Universal Robots URScript: quanser_2_150.script

def initialization():
	global program_counter = 1
end
def main():
	first_trajectory_pose = pose_inv(p[0.6, 0.0, 0.617008797653959, -1.20919957615615, 1.20919957615615, -1.20919957615615])
	starting_pose_tcp = get_actual_tcp_pose()
	counter = 0
while(counter < program_counter):
	movel(pose_trans(starting_pose_tcp, pose_trans(first_trajectory_pose,p[0.55, 0.0, 0.617008797653959, -1.20919957615615, 1.20919957615615, -1.20919957615615])), r=0.0)
	movel(pose_trans(starting_pose_tcp, pose_trans(first_trajectory_pose,p[0.55, 0.00146627565982405, 0.401466275659824, -1.20919957615615, 1.20919957615615, -1.20919957615615])), r=0.0)
	movel(pose_trans(starting_pose_tcp, pose_trans(first_trajectory_pose,p[0.6, 0.00146627565982405, 0.401466275659824, -1.20919957615615, 1.20919957615615, -1.20919957615615])), r=0.0)
	movel(pose_trans(starting_pose_tcp, pose_trans(first_trajectory_pose,p[0.6, 0.00879765395894428, 0.401466275659824, -1.20919957615615, 1.20919957615615, -1.20919957615615])), r=0.0)
	movel(pose_trans(starting_pose_tcp, pose_trans(first_trajectory_pose,p[0.6, 0.0161290322580645, 0.401466275659824, -1.20919957615615, 1.20919957615615, -1.20919957615615])), r=0.0)
	movel(pose_trans(starting_pose_tcp, pose_trans(first_trajectory_pose,p[0.6, 0.0234604105571848, 0.401466275659824, -1.20919957615615, 1.20919957615615, -1.20919957615615])), r=0.0)
	movel(pose_trans(starting_pose_tcp, pose_trans(first_trajectory_pose,p[0.6, 0.030791788856305, 0.401466275659824, -1.20919957615615, 1.20919957615615, -1.20919957615615])), r=0.0)
	movel(pose_trans(starting_pose_tcp, pose_trans(first_trajectory_pose,p[0.6, 0.0381231671554252, 0.401466275659824, -1.20919957615615, 1.20919957615615, -1.20919957615615])), r=0.0)
	movel(pose_trans(starting_pose_tcp, pose_trans(first_trajectory_pose,p[0.6, 0.0454545454545455, 0.401466275659824, -1.20919957615615, 1.20919957615615, -1.20919957615615])), r=0.0)
	movel(pose_trans(starting_pose_tcp, pose_trans(first_trajectory_pose,p[0.6, 0.0527859237536657, 0.401466275659824, -1.20919957615615, 1.20919957615615, -1.20919957615615])), r=0.0)
	movel(pose_trans(starting_pose_tcp, pose_trans(first_trajectory_pose,p[0.6, 0.0601173020527859, 0.401466275659824, -1.20919957615615, 1.20919957615615, -1.20919957615615])), r=0.0)
	movel(pose_trans(starting_pose_tcp, pose_trans(first_trajectory_pose,p[0.6, 0.0674486803519062, 0.401466275659824, -1.20919957615615, 1.20919957615615, -1.20919957615615])), r=0.0)
	movel(pose_trans(starting_pose_tcp, pose_trans(first_trajectory_pose,p[0.6, 0.0747800586510264, 0.401466275659824, -1.20919957615615, 1.20919957615615, -1.20919957615615])), r=0.0)
	movel(pose_trans(starting_pose_tcp, pose_trans(first_trajectory_pose,p[0.6, 0.0821114369501466, 0.401466275659824, -1.20919957615615, 1.20919957615615, -1.20919957615615])), r=0.0)
	movel(pose_trans(starting_pose_tcp, pose_trans(first_trajectory_pose,p[0.6, 0.0894428152492669, 0.401466275659824, -1.20919957615615, 1.20919957615615, -1.20919957615615])), r=0.0)
	movel(pose_trans(starting_pose_tcp, pose_trans(first_trajectory_pose,p[0.6, 0.0967741935483871, 0.401466275659824, -1.20919957615615, 1.20919957615615, -1.20919957615615])), r=0.0)
	movel(pose_trans(starting_pose_tcp, pose_trans(first_trajectory_pose,p[0.6, 0.104105571847507, 0.401466275659824, -1.20919957615615, 1.20919957615615, -1.20919957615615])), r=0.0)
	movel(pose_trans(starting_pose_tcp, pose_trans(first_trajectory_pose,p[0.6, 0.111436950146628, 0.401466275659824, -1.20919957615615, 1.20919957615615, -1.20919957615615])), r=0.0)
	movel(pose_trans(starting_pose_tcp, pose_trans(first_trajectory_pose,p[0.6, 0.118768328445748, 0.401466275659824, -1.20919957615615, 1.20919957615615, -1.20919957615615])), r=0.0)
	movel(pose_trans(starting_pose_tcp, pose_trans(first_trajectory_pose,p[0.6, 0.126099706744868, 0.401466275659824, -1.20919957615615, 1.20919957615615, -1.20919957615615])), r=0.0)
	movel(pose_trans(starting_pose_tcp, pose_trans(first_trajectory_pose,p[0.6, 0.133431085043988, 0.401466275659824, -1.20919957615615, 1.20919957615615, -1.20919957615615])), r=0.0)
	movel(pose_trans(starting_pose_tcp, pose_trans(first_trajectory_pose,p[0.6, 0.140762463343109, 0.401466275659824, -1.20919957615615, 1.20919957615615, -1.20919957615615])), r=0.0)
	movel(pose_trans(starting_pose_tcp, pose_trans(first_trajectory_pose,p[0.6, 0.148093841642229, 0.401466275659824, -1.20919957615615, 1.20919957615615, -1.20919957615615])), r=0.0)
	movel(pose_trans(starting_pose_tcp, pose_trans(first_trajectory_pose,p[0.6, 0.155425219941349, 0.401466275659824, -1.20919957615615, 1.20919957615615, -1.20919957615615])), r=0.0)
	movel(pose_trans(starting_pose_tcp, pose_trans(first_trajectory_pose,p[0.6, 0.162756598240469, 0.401466275659824, -1.20919957615615, 1.20919957615615, -1.20919957615615])), r=0.0)
	movel(pose_trans(starting_pose_tcp, pose_trans(first_trajectory_pose,p[0.6, 0.170087976539589, 0.401466275659824, -1.20919957615615, 1.20919957615615, -1.20919957615615])), r=0.0)
	movel(pose_trans(starting_pose_tcp, pose_trans(first_trajectory_pose,p[0.6, 0.17741935483871, 0.401466275659824, -1.20919957615615, 1.20919957615615, -1.20919957615615])), r=0.0)
	movel(pose_trans(starting_pose_tcp, pose_trans(first_trajectory_pose,p[0.6, 0.18475073313783, 0.401466275659824, -1.20919957615615, 1.20919957615615, -1.20919957615615])), r=0.0)
	movel(pose_trans(starting_pose_tcp, pose_trans(first_trajectory_pose,p[0.6, 0.19208211143695, 0.401466275659824, -1.20919957615615, 1.20919957615615, -1.20919957615615])), r=0.0)
	movel(pose_trans(starting_pose_tcp, pose_trans(first_trajectory_pose,p[0.6, 0.19941348973607, 0.401466275659824, -1.20919957615615, 1.20919957615615, -1.20919957615615])), r=0.0)
	movel(pose_trans(starting_pose_tcp, pose_trans(first_trajectory_pose,p[0.6, 0.206744868035191, 0.401466275659824, -1.20919957615615, 1.20919957615615, -1.20919957615615])), r=0.0)
	movel(pose_trans(starting_pose_tcp, pose_trans(first_trajectory_pose,p[0.6, 0.214076246334311, 0.401466275659824, -1.20919957615615, 1.20919957615615, -1.20919957615615])), r=0.0)
	movel(pose_trans(starting_pose_tcp, pose_trans(first_trajectory_pose,p[0.6, 0.221407624633431, 0.401466275659824, -1.20919957615615, 1.20919957615615, -1.20919957615615])), r=0.0)
	movel(pose_trans(starting_pose_tcp, pose_trans(first_trajectory_pose,p[0.6, 0.228739002932551, 0.401466275659824, -1.20919957615615, 1.20919957615615, -1.20919957615615])), r=0.0)
	movel(pose_trans(starting_pose_tcp, pose_trans(first_trajectory_pose,p[0.6, 0.236070381231672, 0.401466275659824, -1.20919957615615, 1.20919957615615, -1.20919957615615])), r=0.0)
	movel(pose_trans(starting_pose_tcp, pose_trans(first_trajectory_pose,p[0.6, 0.243401759530792, 0.401466275659824, -1.20919957615615, 1.20919957615615, -1.20919957615615])), r=0.0)
	movel(pose_trans(starting_pose_tcp, pose_trans(first_trajectory_pose,p[0.6, 0.250733137829912, 0.401466275659824, -1.20919957615615, 1.20919957615615, -1.20919957615615])), r=0.0)
	movel(pose_trans(starting_pose_tcp, pose_trans(first_trajectory_pose,p[0.6, 0.258064516129032, 0.401466275659824, -1.20919957615615, 1.20919957615615, -1.20919957615615])), r=0.0)
	movel(pose_trans(starting_pose_tcp, pose_trans(first_trajectory_pose,p[0.6, 0.265395894428152, 0.401466275659824, -1.20919957615615, 1.20919957615615, -1.20919957615615])), r=0.0)
	movel(pose_trans(starting_pose_tcp, pose_trans(first_trajectory_pose,p[0.6, 0.272727272727273, 0.401466275659824, -1.20919957615615, 1.20919957615615, -1.20919957615615])), r=0.0)
	movel(pose_trans(starting_pose_tcp, pose_trans(first_trajectory_pose,p[0.6, 0.280058651026393, 0.401466275659824, -1.20919957615615, 1.20919957615615, -1.20919957615615])), r=0.0)
	movel(pose_trans(starting_pose_tcp, pose_trans(first_trajectory_pose,p[0.6, 0.287390029325513, 0.401466275659824, -1.20919957615615, 1.20919957615615, -1.20919957615615])), r=0.0)
	movel(pose_trans(starting_pose_tcp, pose_trans(first_trajectory_pose,p[0.6, 0.294721407624633, 0.401466275659824, -1.20919957615615, 1.20919957615615, -1.20919957615615])), r=0.0)
	movel(pose_trans(starting_pose_tcp, pose_trans(first_trajectory_pose,p[0.6, 0.302052785923754, 0.401466275659824, -1.20919957615615, 1.20919957615615, -1.20919957615615])), r=0.0)
	movel(pose_trans(starting_pose_tcp, pose_trans(first_trajectory_pose,p[0.6, 0.309384164222874, 0.401466275659824, -1.20919957615615, 1.20919957615615, -1.20919957615615])), r=0.0)
	movel(pose_trans(starting_pose_tcp, pose_trans(first_trajectory_pose,p[0.6, 0.316715542521994, 0.401466275659824, -1.20919957615615, 1.20919957615615, -1.20919957615615])), r=0.0)
	movel(pose_trans(starting_pose_tcp, pose_trans(first_trajectory_pose,p[0.6, 0.324046920821114, 0.401466275659824, -1.20919957615615, 1.20919957615615, -1.20919957615615])), r=0.0)
	movel(pose_trans(starting_pose_tcp, pose_trans(first_trajectory_pose,p[0.6, 0.331378299120235, 0.401466275659824, -1.20919957615615, 1.20919957615615, -1.20919957615615])), r=0.0)
	movel(pose_trans(starting_pose_tcp, pose_trans(first_trajectory_pose,p[0.6, 0.338709677419355, 0.401466275659824, -1.20919957615615, 1.20919957615615, -1.20919957615615])), r=0.0)
	movel(pose_trans(starting_pose_tcp, pose_trans(first_trajectory_pose,p[0.6, 0.346041055718475, 0.401466275659824, -1.20919957615615, 1.20919957615615, -1.20919957615615])), r=0.0)
	movel(pose_trans(starting_pose_tcp, pose_trans(first_trajectory_pose,p[0.6, 0.353372434017595, 0.401466275659824, -1.20919957615615, 1.20919957615615, -1.20919957615615])), r=0.0)
	movel(pose_trans(starting_pose_tcp, pose_trans(first_trajectory_pose,p[0.6, 0.360703812316716, 0.401466275659824, -1.20919957615615, 1.20919957615615, -1.20919957615615])), r=0.0)
	movel(pose_trans(starting_pose_tcp, pose_trans(first_trajectory_pose,p[0.6, 0.368035190615836, 0.401466275659824, -1.20919957615615, 1.20919957615615, -1.20919957615615])), r=0.0)
	movel(pose_trans(starting_pose_tcp, pose_trans(first_trajectory_pose,p[0.6, 0.375366568914956, 0.401466275659824, -1.20919957615615, 1.20919957615615, -1.20919957615615])), r=0.0)
	movel(pose_trans(starting_pose_tcp, pose_trans(first_trajectory_pose,p[0.6, 0.382697947214076, 0.401466275659824, -1.20919957615615, 1.20919957615615, -1.20919957615615])), r=0.0)
	movel(pose_trans(starting_pose_tcp, pose_trans(first_trajectory_pose,p[0.6, 0.390029325513196, 0.401466275659824, -1.20919957615615, 1.20919957615615, -1.20919957615615])), r=0.0)
	movel(pose_trans(starting_pose_tcp, pose_trans(first_trajectory_pose,p[0.6, 0.397360703812317, 0.401466275659824, -1.20919957615615, 1.20919957615615, -1.20919957615615])), r=0.0)
	movel(pose_trans(starting_pose_tcp, pose_trans(first_trajectory_pose,p[0.6, 0.404692082111437, 0.401466275659824, -1.20919957615615, 1.20919957615615, -1.20919957615615])), r=0.0)
	movel(pose_trans(starting_pose_tcp, pose_trans(first_trajectory_pose,p[0.6, 0.412023460410557, 0.401466275659824, -1.20919957615615, 1.20919957615615, -1.20919957615615])), r=0.0)
	movel(pose_trans(starting_pose_tcp, pose_trans(first_trajectory_pose,p[0.6, 0.419354838709677, 0.401466275659824, -1.20919957615615, 1.20919957615615, -1.20919957615615])), r=0.0)
	movel(pose_trans(starting_pose_tcp, pose_trans(first_trajectory_pose,p[0.6, 0.426686217008798, 0.401466275659824, -1.20919957615615, 1.20919957615615, -1.20919957615615])), r=0.0)
	movel(pose_trans(starting_pose_tcp, pose_trans(first_trajectory_pose,p[0.6, 0.434017595307918, 0.401466275659824, -1.20919957615615, 1.20919957615615, -1.20919957615615])), r=0.0)
	movel(pose_trans(starting_pose_tcp, pose_trans(first_trajectory_pose,p[0.6, 0.441348973607038, 0.401466275659824, -1.20919957615615, 1.20919957615615, -1.20919957615615])), r=0.0)
	movel(pose_trans(starting_pose_tcp, pose_trans(first_trajectory_pose,p[0.6, 0.448680351906158, 0.401466275659824, -1.20919957615615, 1.20919957615615, -1.20919957615615])), r=0.0)
	movel(pose_trans(starting_pose_tcp, pose_trans(first_trajectory_pose,p[0.6, 0.456011730205279, 0.401466275659824, -1.20919957615615, 1.20919957615615, -1.20919957615615])), r=0.0)
	movel(pose_trans(starting_pose_tcp, pose_trans(first_trajectory_pose,p[0.6, 0.463343108504399, 0.401466275659824, -1.20919957615615, 1.20919957615615, -1.20919957615615])), r=0.0)
	movel(pose_trans(starting_pose_tcp, pose_trans(first_trajectory_pose,p[0.6, 0.470674486803519, 0.401466275659824, -1.20919957615615, 1.20919957615615, -1.20919957615615])), r=0.0)
	movel(pose_trans(starting_pose_tcp, pose_trans(first_trajectory_pose,p[0.6, 0.478005865102639, 0.401466275659824, -1.20919957615615, 1.20919957615615, -1.20919957615615])), r=0.0)
	movel(pose_trans(starting_pose_tcp, pose_trans(first_trajectory_pose,p[0.6, 0.48533724340176, 0.401466275659824, -1.20919957615615, 1.20919957615615, -1.20919957615615])), r=0.0)
	movel(pose_trans(starting_pose_tcp, pose_trans(first_trajectory_pose,p[0.6, 0.49266862170088, 0.401466275659824, -1.20919957615615, 1.20919957615615, -1.20919957615615])), r=0.0)
	movel(pose_trans(starting_pose_tcp, pose_trans(first_trajectory_pose,p[0.6, 0.5, 0.401466275659824, -1.20919957615615, 1.20919957615615, -1.20919957615615])), r=0.0)
	movel(pose_trans(starting_pose_tcp, pose_trans(first_trajectory_pose,p[0.6, 0.5, 0.408797653958944, -1.20919957615615, 1.20919957615615, -1.20919957615615])), r=0.0)
	movel(pose_trans(starting_pose_tcp, pose_trans(first_trajectory_pose,p[0.6, 0.5, 0.416129032258065, -1.20919957615615, 1.20919957615615, -1.20919957615615])), r=0.0)
	movel(pose_trans(starting_pose_tcp, pose_trans(first_trajectory_pose,p[0.6, 0.5, 0.423460410557185, -1.20919957615615, 1.20919957615615, -1.20919957615615])), r=0.0)
	movel(pose_trans(starting_pose_tcp, pose_trans(first_trajectory_pose,p[0.6, 0.5, 0.430791788856305, -1.20919957615615, 1.20919957615615, -1.20919957615615])), r=0.0)
	movel(pose_trans(starting_pose_tcp, pose_trans(first_trajectory_pose,p[0.6, 0.5, 0.438123167155425, -1.20919957615615, 1.20919957615615, -1.20919957615615])), r=0.0)
	movel(pose_trans(starting_pose_tcp, pose_trans(first_trajectory_pose,p[0.6, 0.5, 0.445454545454545, -1.20919957615615, 1.20919957615615, -1.20919957615615])), r=0.0)
	movel(pose_trans(starting_pose_tcp, pose_trans(first_trajectory_pose,p[0.6, 0.5, 0.452785923753666, -1.20919957615615, 1.20919957615615, -1.20919957615615])), r=0.0)
	movel(pose_trans(starting_pose_tcp, pose_trans(first_trajectory_pose,p[0.6, 0.5, 0.460117302052786, -1.20919957615615, 1.20919957615615, -1.20919957615615])), r=0.0)
	movel(pose_trans(starting_pose_tcp, pose_trans(first_trajectory_pose,p[0.6, 0.5, 0.467448680351906, -1.20919957615615, 1.20919957615615, -1.20919957615615])), r=0.0)
	movel(pose_trans(starting_pose_tcp, pose_trans(first_trajectory_pose,p[0.6, 0.5, 0.474780058651026, -1.20919957615615, 1.20919957615615, -1.20919957615615])), r=0.0)
	movel(pose_trans(starting_pose_tcp, pose_trans(first_trajectory_pose,p[0.6, 0.5, 0.482111436950147, -1.20919957615615, 1.20919957615615, -1.20919957615615])), r=0.0)
	movel(pose_trans(starting_pose_tcp, pose_trans(first_trajectory_pose,p[0.6, 0.5, 0.486510263929619, -1.20919957615615, 1.20919957615615, -1.20919957615615])), r=0.0)
	movel(pose_trans(starting_pose_tcp, pose_trans(first_trajectory_pose,p[0.6, 0.498533724340176, 0.479178885630499, -1.20919957615615, 1.20919957615615, -1.20919957615615])), r=0.0)
	movel(pose_trans(starting_pose_tcp, pose_trans(first_trajectory_pose,p[0.6, 0.495601173020528, 0.471847507331378, -1.20919957615615, 1.20919957615615, -1.20919957615615])), r=0.0)
	movel(pose_trans(starting_pose_tcp, pose_trans(first_trajectory_pose,p[0.6, 0.491202346041056, 0.464516129032258, -1.20919957615615, 1.20919957615615, -1.20919957615615])), r=0.0)
	movel(pose_trans(starting_pose_tcp, pose_trans(first_trajectory_pose,p[0.6, 0.486803519061584, 0.457184750733138, -1.20919957615615, 1.20919957615615, -1.20919957615615])), r=0.0)
	movel(pose_trans(starting_pose_tcp, pose_trans(first_trajectory_pose,p[0.6, 0.479472140762463, 0.449853372434018, -1.20919957615615, 1.20919957615615, -1.20919957615615])), r=0.0)
	movel(pose_trans(starting_pose_tcp, pose_trans(first_trajectory_pose,p[0.6, 0.472140762463343, 0.442521994134897, -1.20919957615615, 1.20919957615615, -1.20919957615615])), r=0.0)
	movel(pose_trans(starting_pose_tcp, pose_trans(first_trajectory_pose,p[0.6, 0.464809384164223, 0.436656891495601, -1.20919957615615, 1.20919957615615, -1.20919957615615])), r=0.0)
	movel(pose_trans(starting_pose_tcp, pose_trans(first_trajectory_pose,p[0.6, 0.457478005865103, 0.430791788856305, -1.20919957615615, 1.20919957615615, -1.20919957615615])), r=0.0)
	movel(pose_trans(starting_pose_tcp, pose_trans(first_trajectory_pose,p[0.6, 0.450146627565982, 0.426392961876833, -1.20919957615615, 1.20919957615615, -1.20919957615615])), r=0.0)
	movel(pose_trans(starting_pose_tcp, pose_trans(first_trajectory_pose,p[0.6, 0.442815249266862, 0.421994134897361, -1.20919957615615, 1.20919957615615, -1.20919957615615])), r=0.0)
	movel(pose_trans(starting_pose_tcp, pose_trans(first_trajectory_pose,p[0.6, 0.435483870967742, 0.417595307917889, -1.20919957615615, 1.20919957615615, -1.20919957615615])), r=0.0)
	movel(pose_trans(starting_pose_tcp, pose_trans(first_trajectory_pose,p[0.6, 0.428152492668622, 0.41466275659824, -1.20919957615615, 1.20919957615615, -1.20919957615615])), r=0.0)
	movel(pose_trans(starting_pose_tcp, pose_trans(first_trajectory_pose,p[0.6, 0.420821114369501, 0.410263929618768, -1.20919957615615, 1.20919957615615, -1.20919957615615])), r=0.0)
	movel(pose_trans(starting_pose_tcp, pose_trans(first_trajectory_pose,p[0.6, 0.413489736070381, 0.40733137829912, -1.20919957615615, 1.20919957615615, -1.20919957615615])), r=0.0)
	movel(pose_trans(starting_pose_tcp, pose_trans(first_trajectory_pose,p[0.6, 0.406158357771261, 0.404398826979472, -1.20919957615615, 1.20919957615615, -1.20919957615615])), r=0.0)
	movel(pose_trans(starting_pose_tcp, pose_trans(first_trajectory_pose,p[0.6, 0.404692082111437, 0.40733137829912, -1.20919957615615, 1.20919957615615, -1.20919957615615])), r=0.0)
	movel(pose_trans(starting_pose_tcp, pose_trans(first_trajectory_pose,p[0.6, 0.410557184750733, 0.41466275659824, -1.20919957615615, 1.20919957615615, -1.20919957615615])), r=0.0)
	movel(pose_trans(starting_pose_tcp, pose_trans(first_trajectory_pose,p[0.6, 0.413489736070381, 0.421994134897361, -1.20919957615615, 1.20919957615615, -1.20919957615615])), r=0.0)
	movel(pose_trans(starting_pose_tcp, pose_trans(first_trajectory_pose,p[0.6, 0.416422287390029, 0.429325513196481, -1.20919957615615, 1.20919957615615, -1.20919957615615])), r=0.0)
	movel(pose_trans(starting_pose_tcp, pose_trans(first_trajectory_pose,p[0.6, 0.416422287390029, 0.436656891495601, -1.20919957615615, 1.20919957615615, -1.20919957615615])), r=0.0)
	movel(pose_trans(starting_pose_tcp, pose_trans(first_trajectory_pose,p[0.6, 0.414956011730205, 0.443988269794721, -1.20919957615615, 1.20919957615615, -1.20919957615615])), r=0.0)
	movel(pose_trans(starting_pose_tcp, pose_trans(first_trajectory_pose,p[0.6, 0.409090909090909, 0.451319648093842, -1.20919957615615, 1.20919957615615, -1.20919957615615])), r=0.0)
	movel(pose_trans(starting_pose_tcp, pose_trans(first_trajectory_pose,p[0.6, 0.401759530791789, 0.455718475073314, -1.20919957615615, 1.20919957615615, -1.20919957615615])), r=0.0)
	movel(pose_trans(starting_pose_tcp, pose_trans(first_trajectory_pose,p[0.6, 0.394428152492669, 0.458651026392962, -1.20919957615615, 1.20919957615615, -1.20919957615615])), r=0.0)
	movel(pose_trans(starting_pose_tcp, pose_trans(first_trajectory_pose,p[0.6, 0.387096774193548, 0.458651026392962, -1.20919957615615, 1.20919957615615, -1.20919957615615])), r=0.0)
	movel(pose_trans(starting_pose_tcp, pose_trans(first_trajectory_pose,p[0.6, 0.379765395894428, 0.458651026392962, -1.20919957615615, 1.20919957615615, -1.20919957615615])), r=0.0)
	movel(pose_trans(starting_pose_tcp, pose_trans(first_trajectory_pose,p[0.6, 0.372434017595308, 0.455718475073314, -1.20919957615615, 1.20919957615615, -1.20919957615615])), r=0.0)
	movel(pose_trans(starting_pose_tcp, pose_trans(first_trajectory_pose,p[0.6, 0.365102639296188, 0.452785923753666, -1.20919957615615, 1.20919957615615, -1.20919957615615])), r=0.0)
	movel(pose_trans(starting_pose_tcp, pose_trans(first_trajectory_pose,p[0.6, 0.357771260997067, 0.448387096774194, -1.20919957615615, 1.20919957615615, -1.20919957615615])), r=0.0)
	movel(pose_trans(starting_pose_tcp, pose_trans(first_trajectory_pose,p[0.6, 0.350439882697947, 0.442521994134897, -1.20919957615615, 1.20919957615615, -1.20919957615615])), r=0.0)
	movel(pose_trans(starting_pose_tcp, pose_trans(first_trajectory_pose,p[0.6, 0.343108504398827, 0.443988269794721, -1.20919957615615, 1.20919957615615, -1.20919957615615])), r=0.0)
	movel(pose_trans(starting_pose_tcp, pose_trans(first_trajectory_pose,p[0.6, 0.335777126099707, 0.448387096774194, -1.20919957615615, 1.20919957615615, -1.20919957615615])), r=0.0)
	movel(pose_trans(starting_pose_tcp, pose_trans(first_trajectory_pose,p[0.6, 0.328445747800586, 0.452785923753666, -1.20919957615615, 1.20919957615615, -1.20919957615615])), r=0.0)
	movel(pose_trans(starting_pose_tcp, pose_trans(first_trajectory_pose,p[0.6, 0.321114369501466, 0.455718475073314, -1.20919957615615, 1.20919957615615, -1.20919957615615])), r=0.0)
	movel(pose_trans(starting_pose_tcp, pose_trans(first_trajectory_pose,p[0.6, 0.313782991202346, 0.457184750733138, -1.20919957615615, 1.20919957615615, -1.20919957615615])), r=0.0)
	movel(pose_trans(starting_pose_tcp, pose_trans(first_trajectory_pose,p[0.6, 0.306451612903226, 0.455718475073314, -1.20919957615615, 1.20919957615615, -1.20919957615615])), r=0.0)
	movel(pose_trans(starting_pose_tcp, pose_trans(first_trajectory_pose,p[0.6, 0.299120234604106, 0.452785923753666, -1.20919957615615, 1.20919957615615, -1.20919957615615])), r=0.0)
	movel(pose_trans(starting_pose_tcp, pose_trans(first_trajectory_pose,p[0.6, 0.291788856304985, 0.448387096774194, -1.20919957615615, 1.20919957615615, -1.20919957615615])), r=0.0)
	movel(pose_trans(starting_pose_tcp, pose_trans(first_trajectory_pose,p[0.6, 0.284457478005865, 0.442521994134897, -1.20919957615615, 1.20919957615615, -1.20919957615615])), r=0.0)
	movel(pose_trans(starting_pose_tcp, pose_trans(first_trajectory_pose,p[0.6, 0.277126099706745, 0.435190615835777, -1.20919957615615, 1.20919957615615, -1.20919957615615])), r=0.0)
	movel(pose_trans(starting_pose_tcp, pose_trans(first_trajectory_pose,p[0.6, 0.271260997067449, 0.427859237536657, -1.20919957615615, 1.20919957615615, -1.20919957615615])), r=0.0)
	movel(pose_trans(starting_pose_tcp, pose_trans(first_trajectory_pose,p[0.6, 0.265395894428152, 0.420527859237537, -1.20919957615615, 1.20919957615615, -1.20919957615615])), r=0.0)
	movel(pose_trans(starting_pose_tcp, pose_trans(first_trajectory_pose,p[0.6, 0.259530791788856, 0.413196480938416, -1.20919957615615, 1.20919957615615, -1.20919957615615])), r=0.0)
	movel(pose_trans(starting_pose_tcp, pose_trans(first_trajectory_pose,p[0.6, 0.25366568914956, 0.405865102639296, -1.20919957615615, 1.20919957615615, -1.20919957615615])), r=0.0)
	movel(pose_trans(starting_pose_tcp, pose_trans(first_trajectory_pose,p[0.6, 0.24633431085044, 0.40733137829912, -1.20919957615615, 1.20919957615615, -1.20919957615615])), r=0.0)
	movel(pose_trans(starting_pose_tcp, pose_trans(first_trajectory_pose,p[0.6, 0.241935483870968, 0.41466275659824, -1.20919957615615, 1.20919957615615, -1.20919957615615])), r=0.0)
	movel(pose_trans(starting_pose_tcp, pose_trans(first_trajectory_pose,p[0.6, 0.236070381231672, 0.421994134897361, -1.20919957615615, 1.20919957615615, -1.20919957615615])), r=0.0)
	movel(pose_trans(starting_pose_tcp, pose_trans(first_trajectory_pose,p[0.6, 0.230205278592375, 0.429325513196481, -1.20919957615615, 1.20919957615615, -1.20919957615615])), r=0.0)
	movel(pose_trans(starting_pose_tcp, pose_trans(first_trajectory_pose,p[0.6, 0.222873900293255, 0.436656891495601, -1.20919957615615, 1.20919957615615, -1.20919957615615])), r=0.0)
	movel(pose_trans(starting_pose_tcp, pose_trans(first_trajectory_pose,p[0.6, 0.215542521994135, 0.443988269794721, -1.20919957615615, 1.20919957615615, -1.20919957615615])), r=0.0)
	movel(pose_trans(starting_pose_tcp, pose_trans(first_trajectory_pose,p[0.6, 0.208211143695015, 0.448387096774194, -1.20919957615615, 1.20919957615615, -1.20919957615615])), r=0.0)
	movel(pose_trans(starting_pose_tcp, pose_trans(first_trajectory_pose,p[0.6, 0.200879765395894, 0.452785923753666, -1.20919957615615, 1.20919957615615, -1.20919957615615])), r=0.0)
	movel(pose_trans(starting_pose_tcp, pose_trans(first_trajectory_pose,p[0.6, 0.193548387096774, 0.455718475073314, -1.20919957615615, 1.20919957615615, -1.20919957615615])), r=0.0)
	movel(pose_trans(starting_pose_tcp, pose_trans(first_trajectory_pose,p[0.6, 0.186217008797654, 0.457184750733138, -1.20919957615615, 1.20919957615615, -1.20919957615615])), r=0.0)
	movel(pose_trans(starting_pose_tcp, pose_trans(first_trajectory_pose,p[0.6, 0.178885630498534, 0.455718475073314, -1.20919957615615, 1.20919957615615, -1.20919957615615])), r=0.0)
	movel(pose_trans(starting_pose_tcp, pose_trans(first_trajectory_pose,p[0.6, 0.171554252199413, 0.452785923753666, -1.20919957615615, 1.20919957615615, -1.20919957615615])), r=0.0)
	movel(pose_trans(starting_pose_tcp, pose_trans(first_trajectory_pose,p[0.6, 0.164222873900293, 0.448387096774194, -1.20919957615615, 1.20919957615615, -1.20919957615615])), r=0.0)
	movel(pose_trans(starting_pose_tcp, pose_trans(first_trajectory_pose,p[0.6, 0.156891495601173, 0.442521994134897, -1.20919957615615, 1.20919957615615, -1.20919957615615])), r=0.0)
	movel(pose_trans(starting_pose_tcp, pose_trans(first_trajectory_pose,p[0.6, 0.149560117302053, 0.443988269794721, -1.20919957615615, 1.20919957615615, -1.20919957615615])), r=0.0)
	movel(pose_trans(starting_pose_tcp, pose_trans(first_trajectory_pose,p[0.6, 0.142228739002933, 0.449853372434018, -1.20919957615615, 1.20919957615615, -1.20919957615615])), r=0.0)
	movel(pose_trans(starting_pose_tcp, pose_trans(first_trajectory_pose,p[0.6, 0.134897360703812, 0.45425219941349, -1.20919957615615, 1.20919957615615, -1.20919957615615])), r=0.0)
	movel(pose_trans(starting_pose_tcp, pose_trans(first_trajectory_pose,p[0.6, 0.127565982404692, 0.457184750733138, -1.20919957615615, 1.20919957615615, -1.20919957615615])), r=0.0)
	movel(pose_trans(starting_pose_tcp, pose_trans(first_trajectory_pose,p[0.6, 0.120234604105572, 0.458651026392962, -1.20919957615615, 1.20919957615615, -1.20919957615615])), r=0.0)
	movel(pose_trans(starting_pose_tcp, pose_trans(first_trajectory_pose,p[0.6, 0.112903225806452, 0.458651026392962, -1.20919957615615, 1.20919957615615, -1.20919957615615])), r=0.0)
	movel(pose_trans(starting_pose_tcp, pose_trans(first_trajectory_pose,p[0.6, 0.105571847507331, 0.457184750733138, -1.20919957615615, 1.20919957615615, -1.20919957615615])), r=0.0)
	movel(pose_trans(starting_pose_tcp, pose_trans(first_trajectory_pose,p[0.6, 0.0982404692082111, 0.455718475073314, -1.20919957615615, 1.20919957615615, -1.20919957615615])), r=0.0)
	movel(pose_trans(starting_pose_tcp, pose_trans(first_trajectory_pose,p[0.6, 0.0909090909090909, 0.449853372434018, -1.20919957615615, 1.20919957615615, -1.20919957615615])), r=0.0)
	movel(pose_trans(starting_pose_tcp, pose_trans(first_trajectory_pose,p[0.6, 0.0865102639296188, 0.442521994134897, -1.20919957615615, 1.20919957615615, -1.20919957615615])), r=0.0)
	movel(pose_trans(starting_pose_tcp, pose_trans(first_trajectory_pose,p[0.6, 0.0850439882697947, 0.435190615835777, -1.20919957615615, 1.20919957615615, -1.20919957615615])), r=0.0)
	movel(pose_trans(starting_pose_tcp, pose_trans(first_trajectory_pose,p[0.6, 0.0850439882697947, 0.427859237536657, -1.20919957615615, 1.20919957615615, -1.20919957615615])), r=0.0)
	movel(pose_trans(starting_pose_tcp, pose_trans(first_trajectory_pose,p[0.6, 0.0879765395894428, 0.420527859237537, -1.20919957615615, 1.20919957615615, -1.20919957615615])), r=0.0)
	movel(pose_trans(starting_pose_tcp, pose_trans(first_trajectory_pose,p[0.6, 0.092375366568915, 0.413196480938416, -1.20919957615615, 1.20919957615615, -1.20919957615615])), r=0.0)
	movel(pose_trans(starting_pose_tcp, pose_trans(first_trajectory_pose,p[0.6, 0.0982404692082111, 0.405865102639296, -1.20919957615615, 1.20919957615615, -1.20919957615615])), r=0.0)
	movel(pose_trans(starting_pose_tcp, pose_trans(first_trajectory_pose,p[0.6, 0.093841642228739, 0.404398826979472, -1.20919957615615, 1.20919957615615, -1.20919957615615])), r=0.0)
	movel(pose_trans(starting_pose_tcp, pose_trans(first_trajectory_pose,p[0.6, 0.0865102639296188, 0.40733137829912, -1.20919957615615, 1.20919957615615, -1.20919957615615])), r=0.0)
	movel(pose_trans(starting_pose_tcp, pose_trans(first_trajectory_pose,p[0.6, 0.0791788856304985, 0.411730205278592, -1.20919957615615, 1.20919957615615, -1.20919957615615])), r=0.0)
	movel(pose_trans(starting_pose_tcp, pose_trans(first_trajectory_pose,p[0.6, 0.0718475073313783, 0.41466275659824, -1.20919957615615, 1.20919957615615, -1.20919957615615])), r=0.0)
	movel(pose_trans(starting_pose_tcp, pose_trans(first_trajectory_pose,p[0.6, 0.0645161290322581, 0.419061583577713, -1.20919957615615, 1.20919957615615, -1.20919957615615])), r=0.0)
	movel(pose_trans(starting_pose_tcp, pose_trans(first_trajectory_pose,p[0.6, 0.0571847507331378, 0.421994134897361, -1.20919957615615, 1.20919957615615, -1.20919957615615])), r=0.0)
	movel(pose_trans(starting_pose_tcp, pose_trans(first_trajectory_pose,p[0.6, 0.0498533724340176, 0.427859237536657, -1.20919957615615, 1.20919957615615, -1.20919957615615])), r=0.0)
	movel(pose_trans(starting_pose_tcp, pose_trans(first_trajectory_pose,p[0.6, 0.0425219941348974, 0.432258064516129, -1.20919957615615, 1.20919957615615, -1.20919957615615])), r=0.0)
	movel(pose_trans(starting_pose_tcp, pose_trans(first_trajectory_pose,p[0.6, 0.0351906158357771, 0.438123167155425, -1.20919957615615, 1.20919957615615, -1.20919957615615])), r=0.0)
	movel(pose_trans(starting_pose_tcp, pose_trans(first_trajectory_pose,p[0.6, 0.0278592375366569, 0.443988269794721, -1.20919957615615, 1.20919957615615, -1.20919957615615])), r=0.0)
	movel(pose_trans(starting_pose_tcp, pose_trans(first_trajectory_pose,p[0.6, 0.0205278592375367, 0.451319648093842, -1.20919957615615, 1.20919957615615, -1.20919957615615])), r=0.0)
	movel(pose_trans(starting_pose_tcp, pose_trans(first_trajectory_pose,p[0.6, 0.0131964809384164, 0.458651026392962, -1.20919957615615, 1.20919957615615, -1.20919957615615])), r=0.0)
	movel(pose_trans(starting_pose_tcp, pose_trans(first_trajectory_pose,p[0.6, 0.00879765395894428, 0.465982404692082, -1.20919957615615, 1.20919957615615, -1.20919957615615])), r=0.0)
	movel(pose_trans(starting_pose_tcp, pose_trans(first_trajectory_pose,p[0.6, 0.00439882697947214, 0.473313782991202, -1.20919957615615, 1.20919957615615, -1.20919957615615])), r=0.0)
	movel(pose_trans(starting_pose_tcp, pose_trans(first_trajectory_pose,p[0.6, 0.00146627565982405, 0.480645161290323, -1.20919957615615, 1.20919957615615, -1.20919957615615])), r=0.0)
	movel(pose_trans(starting_pose_tcp, pose_trans(first_trajectory_pose,p[0.6, 0.00146627565982405, 0.485043988269795, -1.20919957615615, 1.20919957615615, -1.20919957615615])), r=0.0)
	movel(pose_trans(starting_pose_tcp, pose_trans(first_trajectory_pose,p[0.6, 0.00146627565982405, 0.477712609970674, -1.20919957615615, 1.20919957615615, -1.20919957615615])), r=0.0)
	movel(pose_trans(starting_pose_tcp, pose_trans(first_trajectory_pose,p[0.6, 0.00146627565982405, 0.470381231671554, -1.20919957615615, 1.20919957615615, -1.20919957615615])), r=0.0)
	movel(pose_trans(starting_pose_tcp, pose_trans(first_trajectory_pose,p[0.6, 0.00146627565982405, 0.463049853372434, -1.20919957615615, 1.20919957615615, -1.20919957615615])), r=0.0)
	movel(pose_trans(starting_pose_tcp, pose_trans(first_trajectory_pose,p[0.6, 0.00146627565982405, 0.455718475073314, -1.20919957615615, 1.20919957615615, -1.20919957615615])), r=0.0)
	movel(pose_trans(starting_pose_tcp, pose_trans(first_trajectory_pose,p[0.6, 0.00146627565982405, 0.448387096774194, -1.20919957615615, 1.20919957615615, -1.20919957615615])), r=0.0)
	movel(pose_trans(starting_pose_tcp, pose_trans(first_trajectory_pose,p[0.6, 0.00146627565982405, 0.441055718475073, -1.20919957615615, 1.20919957615615, -1.20919957615615])), r=0.0)
	movel(pose_trans(starting_pose_tcp, pose_trans(first_trajectory_pose,p[0.6, 0.00146627565982405, 0.433724340175953, -1.20919957615615, 1.20919957615615, -1.20919957615615])), r=0.0)
	movel(pose_trans(starting_pose_tcp, pose_trans(first_trajectory_pose,p[0.6, 0.00146627565982405, 0.426392961876833, -1.20919957615615, 1.20919957615615, -1.20919957615615])), r=0.0)
	movel(pose_trans(starting_pose_tcp, pose_trans(first_trajectory_pose,p[0.6, 0.00146627565982405, 0.419061583577713, -1.20919957615615, 1.20919957615615, -1.20919957615615])), r=0.0)
	movel(pose_trans(starting_pose_tcp, pose_trans(first_trajectory_pose,p[0.6, 0.00146627565982405, 0.411730205278592, -1.20919957615615, 1.20919957615615, -1.20919957615615])), r=0.0)
	movel(pose_trans(starting_pose_tcp, pose_trans(first_trajectory_pose,p[0.6, 0.00146627565982405, 0.404398826979472, -1.20919957615615, 1.20919957615615, -1.20919957615615])), r=0.0)
	movel(pose_trans(starting_pose_tcp, pose_trans(first_trajectory_pose,p[0.6, 0.00146627565982405, 0.401466275659824, -1.20919957615615, 1.20919957615615, -1.20919957615615])), r=0.0)
	movel(pose_trans(starting_pose_tcp, pose_trans(first_trajectory_pose,p[0.55, 0.00146627565982405, 0.401466275659824, -1.20919957615615, 1.20919957615615, -1.20919957615615])), r=0.0)
	movel(pose_trans(starting_pose_tcp, pose_trans(first_trajectory_pose,p[0.55, 0.00146627565982405, 0.502639296187683, -1.20919957615615, 1.20919957615615, -1.20919957615615])), r=0.0)
	movel(pose_trans(starting_pose_tcp, pose_trans(first_trajectory_pose,p[0.6, 0.00146627565982405, 0.502639296187683, -1.20919957615615, 1.20919957615615, -1.20919957615615])), r=0.0)
	movel(pose_trans(starting_pose_tcp, pose_trans(first_trajectory_pose,p[0.6, 0.00293255131964809, 0.509970674486804, -1.20919957615615, 1.20919957615615, -1.20919957615615])), r=0.0)
	movel(pose_trans(starting_pose_tcp, pose_trans(first_trajectory_pose,p[0.6, 0.00439882697947214, 0.517302052785924, -1.20919957615615, 1.20919957615615, -1.20919957615615])), r=0.0)
	movel(pose_trans(starting_pose_tcp, pose_trans(first_trajectory_pose,p[0.6, 0.00879765395894428, 0.524633431085044, -1.20919957615615, 1.20919957615615, -1.20919957615615])), r=0.0)
	movel(pose_trans(starting_pose_tcp, pose_trans(first_trajectory_pose,p[0.6, 0.0131964809384164, 0.531964809384164, -1.20919957615615, 1.20919957615615, -1.20919957615615])), r=0.0)
	movel(pose_trans(starting_pose_tcp, pose_trans(first_trajectory_pose,p[0.6, 0.0190615835777126, 0.539296187683284, -1.20919957615615, 1.20919957615615, -1.20919957615615])), r=0.0)
	movel(pose_trans(starting_pose_tcp, pose_trans(first_trajectory_pose,p[0.6, 0.0263929618768328, 0.546627565982405, -1.20919957615615, 1.20919957615615, -1.20919957615615])), r=0.0)
	movel(pose_trans(starting_pose_tcp, pose_trans(first_trajectory_pose,p[0.6, 0.032258064516129, 0.552492668621701, -1.20919957615615, 1.20919957615615, -1.20919957615615])), r=0.0)
	movel(pose_trans(starting_pose_tcp, pose_trans(first_trajectory_pose,p[0.6, 0.0395894428152493, 0.559824046920821, -1.20919957615615, 1.20919957615615, -1.20919957615615])), r=0.0)
	movel(pose_trans(starting_pose_tcp, pose_trans(first_trajectory_pose,p[0.6, 0.0469208211143695, 0.565689149560117, -1.20919957615615, 1.20919957615615, -1.20919957615615])), r=0.0)
	movel(pose_trans(starting_pose_tcp, pose_trans(first_trajectory_pose,p[0.6, 0.0542521994134897, 0.570087976539589, -1.20919957615615, 1.20919957615615, -1.20919957615615])), r=0.0)
	movel(pose_trans(starting_pose_tcp, pose_trans(first_trajectory_pose,p[0.6, 0.06158357771261, 0.574486803519062, -1.20919957615615, 1.20919957615615, -1.20919957615615])), r=0.0)
	movel(pose_trans(starting_pose_tcp, pose_trans(first_trajectory_pose,p[0.6, 0.0689149560117302, 0.578885630498534, -1.20919957615615, 1.20919957615615, -1.20919957615615])), r=0.0)
	movel(pose_trans(starting_pose_tcp, pose_trans(first_trajectory_pose,p[0.6, 0.0762463343108504, 0.583284457478006, -1.20919957615615, 1.20919957615615, -1.20919957615615])), r=0.0)
	movel(pose_trans(starting_pose_tcp, pose_trans(first_trajectory_pose,p[0.6, 0.0835777126099707, 0.587683284457478, -1.20919957615615, 1.20919957615615, -1.20919957615615])), r=0.0)
	movel(pose_trans(starting_pose_tcp, pose_trans(first_trajectory_pose,p[0.6, 0.0909090909090909, 0.590615835777126, -1.20919957615615, 1.20919957615615, -1.20919957615615])), r=0.0)
	movel(pose_trans(starting_pose_tcp, pose_trans(first_trajectory_pose,p[0.6, 0.0982404692082111, 0.593548387096774, -1.20919957615615, 1.20919957615615, -1.20919957615615])), r=0.0)
	movel(pose_trans(starting_pose_tcp, pose_trans(first_trajectory_pose,p[0.6, 0.105571847507331, 0.596480938416422, -1.20919957615615, 1.20919957615615, -1.20919957615615])), r=0.0)
	movel(pose_trans(starting_pose_tcp, pose_trans(first_trajectory_pose,p[0.6, 0.112903225806452, 0.59941348973607, -1.20919957615615, 1.20919957615615, -1.20919957615615])), r=0.0)
	movel(pose_trans(starting_pose_tcp, pose_trans(first_trajectory_pose,p[0.6, 0.120234604105572, 0.600879765395894, -1.20919957615615, 1.20919957615615, -1.20919957615615])), r=0.0)
	movel(pose_trans(starting_pose_tcp, pose_trans(first_trajectory_pose,p[0.6, 0.127565982404692, 0.603812316715543, -1.20919957615615, 1.20919957615615, -1.20919957615615])), r=0.0)
	movel(pose_trans(starting_pose_tcp, pose_trans(first_trajectory_pose,p[0.6, 0.134897360703812, 0.602346041055718, -1.20919957615615, 1.20919957615615, -1.20919957615615])), r=0.0)
	movel(pose_trans(starting_pose_tcp, pose_trans(first_trajectory_pose,p[0.6, 0.131964809384164, 0.595014662756598, -1.20919957615615, 1.20919957615615, -1.20919957615615])), r=0.0)
	movel(pose_trans(starting_pose_tcp, pose_trans(first_trajectory_pose,p[0.6, 0.129032258064516, 0.587683284457478, -1.20919957615615, 1.20919957615615, -1.20919957615615])), r=0.0)
	movel(pose_trans(starting_pose_tcp, pose_trans(first_trajectory_pose,p[0.6, 0.129032258064516, 0.580351906158358, -1.20919957615615, 1.20919957615615, -1.20919957615615])), r=0.0)
	movel(pose_trans(starting_pose_tcp, pose_trans(first_trajectory_pose,p[0.6, 0.129032258064516, 0.573020527859238, -1.20919957615615, 1.20919957615615, -1.20919957615615])), r=0.0)
	movel(pose_trans(starting_pose_tcp, pose_trans(first_trajectory_pose,p[0.6, 0.13049853372434, 0.565689149560117, -1.20919957615615, 1.20919957615615, -1.20919957615615])), r=0.0)
	movel(pose_trans(starting_pose_tcp, pose_trans(first_trajectory_pose,p[0.6, 0.133431085043988, 0.558357771260997, -1.20919957615615, 1.20919957615615, -1.20919957615615])), r=0.0)
	movel(pose_trans(starting_pose_tcp, pose_trans(first_trajectory_pose,p[0.6, 0.13782991202346, 0.551026392961877, -1.20919957615615, 1.20919957615615, -1.20919957615615])), r=0.0)
	movel(pose_trans(starting_pose_tcp, pose_trans(first_trajectory_pose,p[0.6, 0.145161290322581, 0.546627565982405, -1.20919957615615, 1.20919957615615, -1.20919957615615])), r=0.0)
	movel(pose_trans(starting_pose_tcp, pose_trans(first_trajectory_pose,p[0.6, 0.152492668621701, 0.542228739002933, -1.20919957615615, 1.20919957615615, -1.20919957615615])), r=0.0)
	movel(pose_trans(starting_pose_tcp, pose_trans(first_trajectory_pose,p[0.6, 0.159824046920821, 0.540762463343109, -1.20919957615615, 1.20919957615615, -1.20919957615615])), r=0.0)
	movel(pose_trans(starting_pose_tcp, pose_trans(first_trajectory_pose,p[0.6, 0.167155425219941, 0.539296187683284, -1.20919957615615, 1.20919957615615, -1.20919957615615])), r=0.0)
	movel(pose_trans(starting_pose_tcp, pose_trans(first_trajectory_pose,p[0.6, 0.174486803519062, 0.539296187683284, -1.20919957615615, 1.20919957615615, -1.20919957615615])), r=0.0)
	movel(pose_trans(starting_pose_tcp, pose_trans(first_trajectory_pose,p[0.6, 0.181818181818182, 0.539296187683284, -1.20919957615615, 1.20919957615615, -1.20919957615615])), r=0.0)
	movel(pose_trans(starting_pose_tcp, pose_trans(first_trajectory_pose,p[0.6, 0.189149560117302, 0.540762463343109, -1.20919957615615, 1.20919957615615, -1.20919957615615])), r=0.0)
	movel(pose_trans(starting_pose_tcp, pose_trans(first_trajectory_pose,p[0.6, 0.196480938416422, 0.542228739002933, -1.20919957615615, 1.20919957615615, -1.20919957615615])), r=0.0)
	movel(pose_trans(starting_pose_tcp, pose_trans(first_trajectory_pose,p[0.6, 0.203812316715543, 0.545161290322581, -1.20919957615615, 1.20919957615615, -1.20919957615615])), r=0.0)
	movel(pose_trans(starting_pose_tcp, pose_trans(first_trajectory_pose,p[0.6, 0.211143695014663, 0.549560117302053, -1.20919957615615, 1.20919957615615, -1.20919957615615])), r=0.0)
	movel(pose_trans(starting_pose_tcp, pose_trans(first_trajectory_pose,p[0.6, 0.218475073313783, 0.556891495601173, -1.20919957615615, 1.20919957615615, -1.20919957615615])), r=0.0)
	movel(pose_trans(starting_pose_tcp, pose_trans(first_trajectory_pose,p[0.6, 0.221407624633431, 0.564222873900293, -1.20919957615615, 1.20919957615615, -1.20919957615615])), r=0.0)
	movel(pose_trans(starting_pose_tcp, pose_trans(first_trajectory_pose,p[0.6, 0.222873900293255, 0.571554252199413, -1.20919957615615, 1.20919957615615, -1.20919957615615])), r=0.0)
	movel(pose_trans(starting_pose_tcp, pose_trans(first_trajectory_pose,p[0.6, 0.222873900293255, 0.578885630498534, -1.20919957615615, 1.20919957615615, -1.20919957615615])), r=0.0)
	movel(pose_trans(starting_pose_tcp, pose_trans(first_trajectory_pose,p[0.6, 0.222873900293255, 0.586217008797654, -1.20919957615615, 1.20919957615615, -1.20919957615615])), r=0.0)
	movel(pose_trans(starting_pose_tcp, pose_trans(first_trajectory_pose,p[0.6, 0.222873900293255, 0.593548387096774, -1.20919957615615, 1.20919957615615, -1.20919957615615])), r=0.0)
	movel(pose_trans(starting_pose_tcp, pose_trans(first_trajectory_pose,p[0.6, 0.222873900293255, 0.600879765395894, -1.20919957615615, 1.20919957615615, -1.20919957615615])), r=0.0)
	movel(pose_trans(starting_pose_tcp, pose_trans(first_trajectory_pose,p[0.6, 0.222873900293255, 0.608211143695015, -1.20919957615615, 1.20919957615615, -1.20919957615615])), r=0.0)
	movel(pose_trans(starting_pose_tcp, pose_trans(first_trajectory_pose,p[0.6, 0.222873900293255, 0.615542521994135, -1.20919957615615, 1.20919957615615, -1.20919957615615])), r=0.0)
	movel(pose_trans(starting_pose_tcp, pose_trans(first_trajectory_pose,p[0.6, 0.227272727272727, 0.611143695014663, -1.20919957615615, 1.20919957615615, -1.20919957615615])), r=0.0)
	movel(pose_trans(starting_pose_tcp, pose_trans(first_trajectory_pose,p[0.6, 0.231671554252199, 0.603812316715543, -1.20919957615615, 1.20919957615615, -1.20919957615615])), r=0.0)
	movel(pose_trans(starting_pose_tcp, pose_trans(first_trajectory_pose,p[0.6, 0.236070381231672, 0.596480938416422, -1.20919957615615, 1.20919957615615, -1.20919957615615])), r=0.0)
	movel(pose_trans(starting_pose_tcp, pose_trans(first_trajectory_pose,p[0.6, 0.240469208211144, 0.590615835777126, -1.20919957615615, 1.20919957615615, -1.20919957615615])), r=0.0)
	movel(pose_trans(starting_pose_tcp, pose_trans(first_trajectory_pose,p[0.6, 0.247800586510264, 0.593548387096774, -1.20919957615615, 1.20919957615615, -1.20919957615615])), r=0.0)
	movel(pose_trans(starting_pose_tcp, pose_trans(first_trajectory_pose,p[0.6, 0.255131964809384, 0.59208211143695, -1.20919957615615, 1.20919957615615, -1.20919957615615])), r=0.0)
	movel(pose_trans(starting_pose_tcp, pose_trans(first_trajectory_pose,p[0.6, 0.262463343108504, 0.590615835777126, -1.20919957615615, 1.20919957615615, -1.20919957615615])), r=0.0)
	movel(pose_trans(starting_pose_tcp, pose_trans(first_trajectory_pose,p[0.6, 0.266862170087977, 0.597947214076246, -1.20919957615615, 1.20919957615615, -1.20919957615615])), r=0.0)
	movel(pose_trans(starting_pose_tcp, pose_trans(first_trajectory_pose,p[0.6, 0.269794721407625, 0.605278592375367, -1.20919957615615, 1.20919957615615, -1.20919957615615])), r=0.0)
	movel(pose_trans(starting_pose_tcp, pose_trans(first_trajectory_pose,p[0.6, 0.274193548387097, 0.612609970674487, -1.20919957615615, 1.20919957615615, -1.20919957615615])), r=0.0)
	movel(pose_trans(starting_pose_tcp, pose_trans(first_trajectory_pose,p[0.6, 0.278592375366569, 0.614076246334311, -1.20919957615615, 1.20919957615615, -1.20919957615615])), r=0.0)
	movel(pose_trans(starting_pose_tcp, pose_trans(first_trajectory_pose,p[0.6, 0.278592375366569, 0.606744868035191, -1.20919957615615, 1.20919957615615, -1.20919957615615])), r=0.0)
	movel(pose_trans(starting_pose_tcp, pose_trans(first_trajectory_pose,p[0.6, 0.278592375366569, 0.59941348973607, -1.20919957615615, 1.20919957615615, -1.20919957615615])), r=0.0)
	movel(pose_trans(starting_pose_tcp, pose_trans(first_trajectory_pose,p[0.6, 0.278592375366569, 0.59208211143695, -1.20919957615615, 1.20919957615615, -1.20919957615615])), r=0.0)
	movel(pose_trans(starting_pose_tcp, pose_trans(first_trajectory_pose,p[0.6, 0.278592375366569, 0.58475073313783, -1.20919957615615, 1.20919957615615, -1.20919957615615])), r=0.0)
	movel(pose_trans(starting_pose_tcp, pose_trans(first_trajectory_pose,p[0.6, 0.278592375366569, 0.57741935483871, -1.20919957615615, 1.20919957615615, -1.20919957615615])), r=0.0)
	movel(pose_trans(starting_pose_tcp, pose_trans(first_trajectory_pose,p[0.6, 0.278592375366569, 0.570087976539589, -1.20919957615615, 1.20919957615615, -1.20919957615615])), r=0.0)
	movel(pose_trans(starting_pose_tcp, pose_trans(first_trajectory_pose,p[0.6, 0.280058651026393, 0.562756598240469, -1.20919957615615, 1.20919957615615, -1.20919957615615])), r=0.0)
	movel(pose_trans(starting_pose_tcp, pose_trans(first_trajectory_pose,p[0.6, 0.284457478005865, 0.555425219941349, -1.20919957615615, 1.20919957615615, -1.20919957615615])), r=0.0)
	movel(pose_trans(starting_pose_tcp, pose_trans(first_trajectory_pose,p[0.6, 0.291788856304985, 0.549560117302053, -1.20919957615615, 1.20919957615615, -1.20919957615615])), r=0.0)
	movel(pose_trans(starting_pose_tcp, pose_trans(first_trajectory_pose,p[0.6, 0.299120234604106, 0.545161290322581, -1.20919957615615, 1.20919957615615, -1.20919957615615])), r=0.0)
	movel(pose_trans(starting_pose_tcp, pose_trans(first_trajectory_pose,p[0.6, 0.306451612903226, 0.542228739002933, -1.20919957615615, 1.20919957615615, -1.20919957615615])), r=0.0)
	movel(pose_trans(starting_pose_tcp, pose_trans(first_trajectory_pose,p[0.6, 0.313782991202346, 0.539296187683284, -1.20919957615615, 1.20919957615615, -1.20919957615615])), r=0.0)
	movel(pose_trans(starting_pose_tcp, pose_trans(first_trajectory_pose,p[0.6, 0.321114369501466, 0.539296187683284, -1.20919957615615, 1.20919957615615, -1.20919957615615])), r=0.0)
	movel(pose_trans(starting_pose_tcp, pose_trans(first_trajectory_pose,p[0.6, 0.328445747800586, 0.539296187683284, -1.20919957615615, 1.20919957615615, -1.20919957615615])), r=0.0)
	movel(pose_trans(starting_pose_tcp, pose_trans(first_trajectory_pose,p[0.6, 0.335777126099707, 0.539296187683284, -1.20919957615615, 1.20919957615615, -1.20919957615615])), r=0.0)
	movel(pose_trans(starting_pose_tcp, pose_trans(first_trajectory_pose,p[0.6, 0.343108504398827, 0.540762463343109, -1.20919957615615, 1.20919957615615, -1.20919957615615])), r=0.0)
	movel(pose_trans(starting_pose_tcp, pose_trans(first_trajectory_pose,p[0.6, 0.350439882697947, 0.543695014662757, -1.20919957615615, 1.20919957615615, -1.20919957615615])), r=0.0)
	movel(pose_trans(starting_pose_tcp, pose_trans(first_trajectory_pose,p[0.6, 0.357771260997067, 0.546627565982405, -1.20919957615615, 1.20919957615615, -1.20919957615615])), r=0.0)
	movel(pose_trans(starting_pose_tcp, pose_trans(first_trajectory_pose,p[0.6, 0.365102639296188, 0.552492668621701, -1.20919957615615, 1.20919957615615, -1.20919957615615])), r=0.0)
	movel(pose_trans(starting_pose_tcp, pose_trans(first_trajectory_pose,p[0.6, 0.36950146627566, 0.559824046920821, -1.20919957615615, 1.20919957615615, -1.20919957615615])), r=0.0)
	movel(pose_trans(starting_pose_tcp, pose_trans(first_trajectory_pose,p[0.6, 0.372434017595308, 0.567155425219941, -1.20919957615615, 1.20919957615615, -1.20919957615615])), r=0.0)
	movel(pose_trans(starting_pose_tcp, pose_trans(first_trajectory_pose,p[0.6, 0.373900293255132, 0.574486803519062, -1.20919957615615, 1.20919957615615, -1.20919957615615])), r=0.0)
	movel(pose_trans(starting_pose_tcp, pose_trans(first_trajectory_pose,p[0.6, 0.372434017595308, 0.581818181818182, -1.20919957615615, 1.20919957615615, -1.20919957615615])), r=0.0)
	movel(pose_trans(starting_pose_tcp, pose_trans(first_trajectory_pose,p[0.6, 0.370967741935484, 0.589149560117302, -1.20919957615615, 1.20919957615615, -1.20919957615615])), r=0.0)
	movel(pose_trans(starting_pose_tcp, pose_trans(first_trajectory_pose,p[0.6, 0.36950146627566, 0.596480938416422, -1.20919957615615, 1.20919957615615, -1.20919957615615])), r=0.0)
	movel(pose_trans(starting_pose_tcp, pose_trans(first_trajectory_pose,p[0.6, 0.368035190615836, 0.603812316715543, -1.20919957615615, 1.20919957615615, -1.20919957615615])), r=0.0)
	movel(pose_trans(starting_pose_tcp, pose_trans(first_trajectory_pose,p[0.6, 0.375366568914956, 0.602346041055718, -1.20919957615615, 1.20919957615615, -1.20919957615615])), r=0.0)
	movel(pose_trans(starting_pose_tcp, pose_trans(first_trajectory_pose,p[0.6, 0.382697947214076, 0.600879765395894, -1.20919957615615, 1.20919957615615, -1.20919957615615])), r=0.0)
	movel(pose_trans(starting_pose_tcp, pose_trans(first_trajectory_pose,p[0.6, 0.390029325513196, 0.59941348973607, -1.20919957615615, 1.20919957615615, -1.20919957615615])), r=0.0)
	movel(pose_trans(starting_pose_tcp, pose_trans(first_trajectory_pose,p[0.6, 0.397360703812317, 0.596480938416422, -1.20919957615615, 1.20919957615615, -1.20919957615615])), r=0.0)
	movel(pose_trans(starting_pose_tcp, pose_trans(first_trajectory_pose,p[0.6, 0.404692082111437, 0.593548387096774, -1.20919957615615, 1.20919957615615, -1.20919957615615])), r=0.0)
	movel(pose_trans(starting_pose_tcp, pose_trans(first_trajectory_pose,p[0.6, 0.412023460410557, 0.590615835777126, -1.20919957615615, 1.20919957615615, -1.20919957615615])), r=0.0)
	movel(pose_trans(starting_pose_tcp, pose_trans(first_trajectory_pose,p[0.6, 0.419354838709677, 0.586217008797654, -1.20919957615615, 1.20919957615615, -1.20919957615615])), r=0.0)
	movel(pose_trans(starting_pose_tcp, pose_trans(first_trajectory_pose,p[0.6, 0.426686217008798, 0.583284457478006, -1.20919957615615, 1.20919957615615, -1.20919957615615])), r=0.0)
	movel(pose_trans(starting_pose_tcp, pose_trans(first_trajectory_pose,p[0.6, 0.434017595307918, 0.578885630498534, -1.20919957615615, 1.20919957615615, -1.20919957615615])), r=0.0)
	movel(pose_trans(starting_pose_tcp, pose_trans(first_trajectory_pose,p[0.6, 0.441348973607038, 0.574486803519062, -1.20919957615615, 1.20919957615615, -1.20919957615615])), r=0.0)
	movel(pose_trans(starting_pose_tcp, pose_trans(first_trajectory_pose,p[0.6, 0.448680351906158, 0.568621700879765, -1.20919957615615, 1.20919957615615, -1.20919957615615])), r=0.0)
	movel(pose_trans(starting_pose_tcp, pose_trans(first_trajectory_pose,p[0.6, 0.456011730205279, 0.564222873900293, -1.20919957615615, 1.20919957615615, -1.20919957615615])), r=0.0)
	movel(pose_trans(starting_pose_tcp, pose_trans(first_trajectory_pose,p[0.6, 0.463343108504399, 0.558357771260997, -1.20919957615615, 1.20919957615615, -1.20919957615615])), r=0.0)
	movel(pose_trans(starting_pose_tcp, pose_trans(first_trajectory_pose,p[0.6, 0.470674486803519, 0.551026392961877, -1.20919957615615, 1.20919957615615, -1.20919957615615])), r=0.0)
	movel(pose_trans(starting_pose_tcp, pose_trans(first_trajectory_pose,p[0.6, 0.478005865102639, 0.545161290322581, -1.20919957615615, 1.20919957615615, -1.20919957615615])), r=0.0)
	movel(pose_trans(starting_pose_tcp, pose_trans(first_trajectory_pose,p[0.6, 0.483870967741935, 0.53782991202346, -1.20919957615615, 1.20919957615615, -1.20919957615615])), r=0.0)
	movel(pose_trans(starting_pose_tcp, pose_trans(first_trajectory_pose,p[0.6, 0.489736070381232, 0.53049853372434, -1.20919957615615, 1.20919957615615, -1.20919957615615])), r=0.0)
	movel(pose_trans(starting_pose_tcp, pose_trans(first_trajectory_pose,p[0.6, 0.494134897360704, 0.52316715542522, -1.20919957615615, 1.20919957615615, -1.20919957615615])), r=0.0)
	movel(pose_trans(starting_pose_tcp, pose_trans(first_trajectory_pose,p[0.6, 0.497067448680352, 0.5158357771261, -1.20919957615615, 1.20919957615615, -1.20919957615615])), r=0.0)
	movel(pose_trans(starting_pose_tcp, pose_trans(first_trajectory_pose,p[0.6, 0.5, 0.50850439882698, -1.20919957615615, 1.20919957615615, -1.20919957615615])), r=0.0)
	movel(pose_trans(starting_pose_tcp, pose_trans(first_trajectory_pose,p[0.6, 0.5, 0.504105571847507, -1.20919957615615, 1.20919957615615, -1.20919957615615])), r=0.0)
	movel(pose_trans(starting_pose_tcp, pose_trans(first_trajectory_pose,p[0.6, 0.5, 0.511436950146628, -1.20919957615615, 1.20919957615615, -1.20919957615615])), r=0.0)
	movel(pose_trans(starting_pose_tcp, pose_trans(first_trajectory_pose,p[0.6, 0.5, 0.518768328445748, -1.20919957615615, 1.20919957615615, -1.20919957615615])), r=0.0)
	movel(pose_trans(starting_pose_tcp, pose_trans(first_trajectory_pose,p[0.6, 0.5, 0.526099706744868, -1.20919957615615, 1.20919957615615, -1.20919957615615])), r=0.0)
	movel(pose_trans(starting_pose_tcp, pose_trans(first_trajectory_pose,p[0.6, 0.5, 0.533431085043988, -1.20919957615615, 1.20919957615615, -1.20919957615615])), r=0.0)
	movel(pose_trans(starting_pose_tcp, pose_trans(first_trajectory_pose,p[0.6, 0.5, 0.540762463343109, -1.20919957615615, 1.20919957615615, -1.20919957615615])), r=0.0)
	movel(pose_trans(starting_pose_tcp, pose_trans(first_trajectory_pose,p[0.6, 0.5, 0.548093841642229, -1.20919957615615, 1.20919957615615, -1.20919957615615])), r=0.0)
	movel(pose_trans(starting_pose_tcp, pose_trans(first_trajectory_pose,p[0.6, 0.5, 0.555425219941349, -1.20919957615615, 1.20919957615615, -1.20919957615615])), r=0.0)
	movel(pose_trans(starting_pose_tcp, pose_trans(first_trajectory_pose,p[0.6, 0.5, 0.562756598240469, -1.20919957615615, 1.20919957615615, -1.20919957615615])), r=0.0)
	movel(pose_trans(starting_pose_tcp, pose_trans(first_trajectory_pose,p[0.6, 0.5, 0.570087976539589, -1.20919957615615, 1.20919957615615, -1.20919957615615])), r=0.0)
	movel(pose_trans(starting_pose_tcp, pose_trans(first_trajectory_pose,p[0.6, 0.5, 0.57741935483871, -1.20919957615615, 1.20919957615615, -1.20919957615615])), r=0.0)
	movel(pose_trans(starting_pose_tcp, pose_trans(first_trajectory_pose,p[0.6, 0.5, 0.58475073313783, -1.20919957615615, 1.20919957615615, -1.20919957615615])), r=0.0)
	movel(pose_trans(starting_pose_tcp, pose_trans(first_trajectory_pose,p[0.6, 0.5, 0.59208211143695, -1.20919957615615, 1.20919957615615, -1.20919957615615])), r=0.0)
	movel(pose_trans(starting_pose_tcp, pose_trans(first_trajectory_pose,p[0.6, 0.5, 0.59941348973607, -1.20919957615615, 1.20919957615615, -1.20919957615615])), r=0.0)
	movel(pose_trans(starting_pose_tcp, pose_trans(first_trajectory_pose,p[0.6, 0.5, 0.606744868035191, -1.20919957615615, 1.20919957615615, -1.20919957615615])), r=0.0)
	movel(pose_trans(starting_pose_tcp, pose_trans(first_trajectory_pose,p[0.6, 0.5, 0.614076246334311, -1.20919957615615, 1.20919957615615, -1.20919957615615])), r=0.0)
	movel(pose_trans(starting_pose_tcp, pose_trans(first_trajectory_pose,p[0.6, 0.495601173020528, 0.617008797653959, -1.20919957615615, 1.20919957615615, -1.20919957615615])), r=0.0)
	movel(pose_trans(starting_pose_tcp, pose_trans(first_trajectory_pose,p[0.6, 0.488269794721408, 0.617008797653959, -1.20919957615615, 1.20919957615615, -1.20919957615615])), r=0.0)
	movel(pose_trans(starting_pose_tcp, pose_trans(first_trajectory_pose,p[0.6, 0.480938416422287, 0.617008797653959, -1.20919957615615, 1.20919957615615, -1.20919957615615])), r=0.0)
	movel(pose_trans(starting_pose_tcp, pose_trans(first_trajectory_pose,p[0.6, 0.473607038123167, 0.617008797653959, -1.20919957615615, 1.20919957615615, -1.20919957615615])), r=0.0)
	movel(pose_trans(starting_pose_tcp, pose_trans(first_trajectory_pose,p[0.6, 0.466275659824047, 0.617008797653959, -1.20919957615615, 1.20919957615615, -1.20919957615615])), r=0.0)
	movel(pose_trans(starting_pose_tcp, pose_trans(first_trajectory_pose,p[0.6, 0.458944281524927, 0.617008797653959, -1.20919957615615, 1.20919957615615, -1.20919957615615])), r=0.0)
	movel(pose_trans(starting_pose_tcp, pose_trans(first_trajectory_pose,p[0.6, 0.451612903225806, 0.617008797653959, -1.20919957615615, 1.20919957615615, -1.20919957615615])), r=0.0)
	movel(pose_trans(starting_pose_tcp, pose_trans(first_trajectory_pose,p[0.6, 0.444281524926686, 0.617008797653959, -1.20919957615615, 1.20919957615615, -1.20919957615615])), r=0.0)
	movel(pose_trans(starting_pose_tcp, pose_trans(first_trajectory_pose,p[0.6, 0.436950146627566, 0.617008797653959, -1.20919957615615, 1.20919957615615, -1.20919957615615])), r=0.0)
	movel(pose_trans(starting_pose_tcp, pose_trans(first_trajectory_pose,p[0.6, 0.429618768328446, 0.617008797653959, -1.20919957615615, 1.20919957615615, -1.20919957615615])), r=0.0)
	movel(pose_trans(starting_pose_tcp, pose_trans(first_trajectory_pose,p[0.6, 0.422287390029326, 0.617008797653959, -1.20919957615615, 1.20919957615615, -1.20919957615615])), r=0.0)
	movel(pose_trans(starting_pose_tcp, pose_trans(first_trajectory_pose,p[0.6, 0.414956011730205, 0.617008797653959, -1.20919957615615, 1.20919957615615, -1.20919957615615])), r=0.0)
	movel(pose_trans(starting_pose_tcp, pose_trans(first_trajectory_pose,p[0.6, 0.407624633431085, 0.617008797653959, -1.20919957615615, 1.20919957615615, -1.20919957615615])), r=0.0)
	movel(pose_trans(starting_pose_tcp, pose_trans(first_trajectory_pose,p[0.6, 0.400293255131965, 0.617008797653959, -1.20919957615615, 1.20919957615615, -1.20919957615615])), r=0.0)
	movel(pose_trans(starting_pose_tcp, pose_trans(first_trajectory_pose,p[0.6, 0.392961876832845, 0.617008797653959, -1.20919957615615, 1.20919957615615, -1.20919957615615])), r=0.0)
	movel(pose_trans(starting_pose_tcp, pose_trans(first_trajectory_pose,p[0.6, 0.385630498533724, 0.617008797653959, -1.20919957615615, 1.20919957615615, -1.20919957615615])), r=0.0)
	movel(pose_trans(starting_pose_tcp, pose_trans(first_trajectory_pose,p[0.6, 0.378299120234604, 0.617008797653959, -1.20919957615615, 1.20919957615615, -1.20919957615615])), r=0.0)
	movel(pose_trans(starting_pose_tcp, pose_trans(first_trajectory_pose,p[0.6, 0.370967741935484, 0.617008797653959, -1.20919957615615, 1.20919957615615, -1.20919957615615])), r=0.0)
	movel(pose_trans(starting_pose_tcp, pose_trans(first_trajectory_pose,p[0.6, 0.363636363636364, 0.617008797653959, -1.20919957615615, 1.20919957615615, -1.20919957615615])), r=0.0)
	movel(pose_trans(starting_pose_tcp, pose_trans(first_trajectory_pose,p[0.6, 0.356304985337243, 0.617008797653959, -1.20919957615615, 1.20919957615615, -1.20919957615615])), r=0.0)
	movel(pose_trans(starting_pose_tcp, pose_trans(first_trajectory_pose,p[0.6, 0.348973607038123, 0.617008797653959, -1.20919957615615, 1.20919957615615, -1.20919957615615])), r=0.0)
	movel(pose_trans(starting_pose_tcp, pose_trans(first_trajectory_pose,p[0.6, 0.341642228739003, 0.617008797653959, -1.20919957615615, 1.20919957615615, -1.20919957615615])), r=0.0)
	movel(pose_trans(starting_pose_tcp, pose_trans(first_trajectory_pose,p[0.6, 0.334310850439883, 0.617008797653959, -1.20919957615615, 1.20919957615615, -1.20919957615615])), r=0.0)
	movel(pose_trans(starting_pose_tcp, pose_trans(first_trajectory_pose,p[0.6, 0.326979472140762, 0.617008797653959, -1.20919957615615, 1.20919957615615, -1.20919957615615])), r=0.0)
	movel(pose_trans(starting_pose_tcp, pose_trans(first_trajectory_pose,p[0.6, 0.319648093841642, 0.617008797653959, -1.20919957615615, 1.20919957615615, -1.20919957615615])), r=0.0)
	movel(pose_trans(starting_pose_tcp, pose_trans(first_trajectory_pose,p[0.6, 0.312316715542522, 0.617008797653959, -1.20919957615615, 1.20919957615615, -1.20919957615615])), r=0.0)
	movel(pose_trans(starting_pose_tcp, pose_trans(first_trajectory_pose,p[0.6, 0.304985337243402, 0.617008797653959, -1.20919957615615, 1.20919957615615, -1.20919957615615])), r=0.0)
	movel(pose_trans(starting_pose_tcp, pose_trans(first_trajectory_pose,p[0.6, 0.297653958944282, 0.617008797653959, -1.20919957615615, 1.20919957615615, -1.20919957615615])), r=0.0)
	movel(pose_trans(starting_pose_tcp, pose_trans(first_trajectory_pose,p[0.6, 0.290322580645161, 0.617008797653959, -1.20919957615615, 1.20919957615615, -1.20919957615615])), r=0.0)
	movel(pose_trans(starting_pose_tcp, pose_trans(first_trajectory_pose,p[0.6, 0.282991202346041, 0.617008797653959, -1.20919957615615, 1.20919957615615, -1.20919957615615])), r=0.0)
	movel(pose_trans(starting_pose_tcp, pose_trans(first_trajectory_pose,p[0.6, 0.275659824046921, 0.617008797653959, -1.20919957615615, 1.20919957615615, -1.20919957615615])), r=0.0)
	movel(pose_trans(starting_pose_tcp, pose_trans(first_trajectory_pose,p[0.6, 0.268328445747801, 0.617008797653959, -1.20919957615615, 1.20919957615615, -1.20919957615615])), r=0.0)
	movel(pose_trans(starting_pose_tcp, pose_trans(first_trajectory_pose,p[0.6, 0.26099706744868, 0.617008797653959, -1.20919957615615, 1.20919957615615, -1.20919957615615])), r=0.0)
	movel(pose_trans(starting_pose_tcp, pose_trans(first_trajectory_pose,p[0.6, 0.25366568914956, 0.617008797653959, -1.20919957615615, 1.20919957615615, -1.20919957615615])), r=0.0)
	movel(pose_trans(starting_pose_tcp, pose_trans(first_trajectory_pose,p[0.6, 0.24633431085044, 0.617008797653959, -1.20919957615615, 1.20919957615615, -1.20919957615615])), r=0.0)
	movel(pose_trans(starting_pose_tcp, pose_trans(first_trajectory_pose,p[0.6, 0.23900293255132, 0.617008797653959, -1.20919957615615, 1.20919957615615, -1.20919957615615])), r=0.0)
	movel(pose_trans(starting_pose_tcp, pose_trans(first_trajectory_pose,p[0.6, 0.231671554252199, 0.617008797653959, -1.20919957615615, 1.20919957615615, -1.20919957615615])), r=0.0)
	movel(pose_trans(starting_pose_tcp, pose_trans(first_trajectory_pose,p[0.6, 0.224340175953079, 0.617008797653959, -1.20919957615615, 1.20919957615615, -1.20919957615615])), r=0.0)
	movel(pose_trans(starting_pose_tcp, pose_trans(first_trajectory_pose,p[0.6, 0.217008797653959, 0.617008797653959, -1.20919957615615, 1.20919957615615, -1.20919957615615])), r=0.0)
	movel(pose_trans(starting_pose_tcp, pose_trans(first_trajectory_pose,p[0.6, 0.209677419354839, 0.617008797653959, -1.20919957615615, 1.20919957615615, -1.20919957615615])), r=0.0)
	movel(pose_trans(starting_pose_tcp, pose_trans(first_trajectory_pose,p[0.6, 0.202346041055718, 0.617008797653959, -1.20919957615615, 1.20919957615615, -1.20919957615615])), r=0.0)
	movel(pose_trans(starting_pose_tcp, pose_trans(first_trajectory_pose,p[0.6, 0.195014662756598, 0.617008797653959, -1.20919957615615, 1.20919957615615, -1.20919957615615])), r=0.0)
	movel(pose_trans(starting_pose_tcp, pose_trans(first_trajectory_pose,p[0.6, 0.187683284457478, 0.617008797653959, -1.20919957615615, 1.20919957615615, -1.20919957615615])), r=0.0)
	movel(pose_trans(starting_pose_tcp, pose_trans(first_trajectory_pose,p[0.6, 0.180351906158358, 0.617008797653959, -1.20919957615615, 1.20919957615615, -1.20919957615615])), r=0.0)
	movel(pose_trans(starting_pose_tcp, pose_trans(first_trajectory_pose,p[0.6, 0.173020527859238, 0.617008797653959, -1.20919957615615, 1.20919957615615, -1.20919957615615])), r=0.0)
	movel(pose_trans(starting_pose_tcp, pose_trans(first_trajectory_pose,p[0.6, 0.165689149560117, 0.617008797653959, -1.20919957615615, 1.20919957615615, -1.20919957615615])), r=0.0)
	movel(pose_trans(starting_pose_tcp, pose_trans(first_trajectory_pose,p[0.6, 0.158357771260997, 0.617008797653959, -1.20919957615615, 1.20919957615615, -1.20919957615615])), r=0.0)
	movel(pose_trans(starting_pose_tcp, pose_trans(first_trajectory_pose,p[0.6, 0.151026392961877, 0.617008797653959, -1.20919957615615, 1.20919957615615, -1.20919957615615])), r=0.0)
	movel(pose_trans(starting_pose_tcp, pose_trans(first_trajectory_pose,p[0.6, 0.143695014662757, 0.617008797653959, -1.20919957615615, 1.20919957615615, -1.20919957615615])), r=0.0)
	movel(pose_trans(starting_pose_tcp, pose_trans(first_trajectory_pose,p[0.6, 0.136363636363636, 0.617008797653959, -1.20919957615615, 1.20919957615615, -1.20919957615615])), r=0.0)
	movel(pose_trans(starting_pose_tcp, pose_trans(first_trajectory_pose,p[0.6, 0.129032258064516, 0.617008797653959, -1.20919957615615, 1.20919957615615, -1.20919957615615])), r=0.0)
	movel(pose_trans(starting_pose_tcp, pose_trans(first_trajectory_pose,p[0.6, 0.121700879765396, 0.617008797653959, -1.20919957615615, 1.20919957615615, -1.20919957615615])), r=0.0)
	movel(pose_trans(starting_pose_tcp, pose_trans(first_trajectory_pose,p[0.6, 0.114369501466276, 0.617008797653959, -1.20919957615615, 1.20919957615615, -1.20919957615615])), r=0.0)
	movel(pose_trans(starting_pose_tcp, pose_trans(first_trajectory_pose,p[0.6, 0.107038123167155, 0.617008797653959, -1.20919957615615, 1.20919957615615, -1.20919957615615])), r=0.0)
	movel(pose_trans(starting_pose_tcp, pose_trans(first_trajectory_pose,p[0.6, 0.0997067448680352, 0.617008797653959, -1.20919957615615, 1.20919957615615, -1.20919957615615])), r=0.0)
	movel(pose_trans(starting_pose_tcp, pose_trans(first_trajectory_pose,p[0.6, 0.092375366568915, 0.617008797653959, -1.20919957615615, 1.20919957615615, -1.20919957615615])), r=0.0)
	movel(pose_trans(starting_pose_tcp, pose_trans(first_trajectory_pose,p[0.6, 0.0850439882697947, 0.617008797653959, -1.20919957615615, 1.20919957615615, -1.20919957615615])), r=0.0)
	movel(pose_trans(starting_pose_tcp, pose_trans(first_trajectory_pose,p[0.6, 0.0777126099706745, 0.617008797653959, -1.20919957615615, 1.20919957615615, -1.20919957615615])), r=0.0)
	movel(pose_trans(starting_pose_tcp, pose_trans(first_trajectory_pose,p[0.6, 0.0703812316715543, 0.617008797653959, -1.20919957615615, 1.20919957615615, -1.20919957615615])), r=0.0)
	movel(pose_trans(starting_pose_tcp, pose_trans(first_trajectory_pose,p[0.6, 0.063049853372434, 0.617008797653959, -1.20919957615615, 1.20919957615615, -1.20919957615615])), r=0.0)
	movel(pose_trans(starting_pose_tcp, pose_trans(first_trajectory_pose,p[0.6, 0.0557184750733138, 0.617008797653959, -1.20919957615615, 1.20919957615615, -1.20919957615615])), r=0.0)
	movel(pose_trans(starting_pose_tcp, pose_trans(first_trajectory_pose,p[0.6, 0.0483870967741935, 0.617008797653959, -1.20919957615615, 1.20919957615615, -1.20919957615615])), r=0.0)
	movel(pose_trans(starting_pose_tcp, pose_trans(first_trajectory_pose,p[0.6, 0.0410557184750733, 0.617008797653959, -1.20919957615615, 1.20919957615615, -1.20919957615615])), r=0.0)
	movel(pose_trans(starting_pose_tcp, pose_trans(first_trajectory_pose,p[0.6, 0.0337243401759531, 0.617008797653959, -1.20919957615615, 1.20919957615615, -1.20919957615615])), r=0.0)
	movel(pose_trans(starting_pose_tcp, pose_trans(first_trajectory_pose,p[0.6, 0.0263929618768328, 0.617008797653959, -1.20919957615615, 1.20919957615615, -1.20919957615615])), r=0.0)
	movel(pose_trans(starting_pose_tcp, pose_trans(first_trajectory_pose,p[0.6, 0.0190615835777126, 0.617008797653959, -1.20919957615615, 1.20919957615615, -1.20919957615615])), r=0.0)
	movel(pose_trans(starting_pose_tcp, pose_trans(first_trajectory_pose,p[0.6, 0.0117302052785924, 0.617008797653959, -1.20919957615615, 1.20919957615615, -1.20919957615615])), r=0.0)
	movel(pose_trans(starting_pose_tcp, pose_trans(first_trajectory_pose,p[0.6, 0.00439882697947214, 0.617008797653959, -1.20919957615615, 1.20919957615615, -1.20919957615615])), r=0.0)
	movel(pose_trans(starting_pose_tcp, pose_trans(first_trajectory_pose,p[0.6, 0.00146627565982405, 0.612609970674487, -1.20919957615615, 1.20919957615615, -1.20919957615615])), r=0.0)
	movel(pose_trans(starting_pose_tcp, pose_trans(first_trajectory_pose,p[0.6, 0.00146627565982405, 0.605278592375367, -1.20919957615615, 1.20919957615615, -1.20919957615615])), r=0.0)
	movel(pose_trans(starting_pose_tcp, pose_trans(first_trajectory_pose,p[0.6, 0.00146627565982405, 0.597947214076246, -1.20919957615615, 1.20919957615615, -1.20919957615615])), r=0.0)
	movel(pose_trans(starting_pose_tcp, pose_trans(first_trajectory_pose,p[0.6, 0.00146627565982405, 0.590615835777126, -1.20919957615615, 1.20919957615615, -1.20919957615615])), r=0.0)
	movel(pose_trans(starting_pose_tcp, pose_trans(first_trajectory_pose,p[0.6, 0.00146627565982405, 0.583284457478006, -1.20919957615615, 1.20919957615615, -1.20919957615615])), r=0.0)
	movel(pose_trans(starting_pose_tcp, pose_trans(first_trajectory_pose,p[0.6, 0.00146627565982405, 0.575953079178886, -1.20919957615615, 1.20919957615615, -1.20919957615615])), r=0.0)
	movel(pose_trans(starting_pose_tcp, pose_trans(first_trajectory_pose,p[0.6, 0.00146627565982405, 0.568621700879765, -1.20919957615615, 1.20919957615615, -1.20919957615615])), r=0.0)
	movel(pose_trans(starting_pose_tcp, pose_trans(first_trajectory_pose,p[0.6, 0.00146627565982405, 0.561290322580645, -1.20919957615615, 1.20919957615615, -1.20919957615615])), r=0.0)
	movel(pose_trans(starting_pose_tcp, pose_trans(first_trajectory_pose,p[0.6, 0.00146627565982405, 0.553958944281525, -1.20919957615615, 1.20919957615615, -1.20919957615615])), r=0.0)
	movel(pose_trans(starting_pose_tcp, pose_trans(first_trajectory_pose,p[0.6, 0.00146627565982405, 0.546627565982405, -1.20919957615615, 1.20919957615615, -1.20919957615615])), r=0.0)
	movel(pose_trans(starting_pose_tcp, pose_trans(first_trajectory_pose,p[0.6, 0.00146627565982405, 0.539296187683284, -1.20919957615615, 1.20919957615615, -1.20919957615615])), r=0.0)
	movel(pose_trans(starting_pose_tcp, pose_trans(first_trajectory_pose,p[0.6, 0.00146627565982405, 0.531964809384164, -1.20919957615615, 1.20919957615615, -1.20919957615615])), r=0.0)
	movel(pose_trans(starting_pose_tcp, pose_trans(first_trajectory_pose,p[0.6, 0.00146627565982405, 0.524633431085044, -1.20919957615615, 1.20919957615615, -1.20919957615615])), r=0.0)
	movel(pose_trans(starting_pose_tcp, pose_trans(first_trajectory_pose,p[0.6, 0.00146627565982405, 0.517302052785924, -1.20919957615615, 1.20919957615615, -1.20919957615615])), r=0.0)
	movel(pose_trans(starting_pose_tcp, pose_trans(first_trajectory_pose,p[0.6, 0.00146627565982405, 0.509970674486804, -1.20919957615615, 1.20919957615615, -1.20919957615615])), r=0.0)
	movel(pose_trans(starting_pose_tcp, pose_trans(first_trajectory_pose,p[0.6, 0.00146627565982405, 0.502639296187683, -1.20919957615615, 1.20919957615615, -1.20919957615615])), r=0.0)
	movel(pose_trans(starting_pose_tcp, pose_trans(first_trajectory_pose,p[0.55, 0.00146627565982405, 0.502639296187683, -1.20919957615615, 1.20919957615615, -1.20919957615615])), r=0.0)
	movel(pose_trans(starting_pose_tcp, pose_trans(first_trajectory_pose,p[0.55, 0, 0.617008797653959, -1.20919957615615, 1.20919957615615, -1.20919957615615])), r=0.0)
	movel(pose_trans(starting_pose_tcp, pose_trans(first_trajectory_pose,p[0.6, 0.0, 0.617008797653959, -1.20919957615615, 1.20919957615615, -1.20919957615615])), r=0.0)
	counter = counter + 1
	end
end
